FUNCTION_BLOCK PAEActValve2_3pos EXTENDS PAEActuator2way_3pos
VAR_INPUT
END_VAR
VAR_OUTPUT
END_VAR
VAR
END_VAR

METHOD PUBLIC PAEActValve2_3pos
VAR_INPUT
END_VAR
END_METHOD

END_FUNCTION_BLOCK

(* stored: Version 1.1.0.1, ProductVersion 3.1.4020.12
   POU PAEActValve2_3pos: Id {7bd99d84-d7d1-4fc7-9615-c23cbe5ddbf2}, SpecialFunc None
   Method PAEActValve2_3pos: Id {8a1fb15d-0692-4d16-9b2a-7e2529212853} *)
